FUNCTION_BLOCK TcoContext_App_1 EXTENDS TcoContext
VAR_INPUT
END_VAR
VAR_OUTPUT
END_VAR
VAR
	ResetToZero : BOOL := TRUE;
	C1	:	LINT	:= 100;
	C2	:	LINT	:= 200;
	TcoObject_Counter_1 : TcoObject_Counter(THIS^);
	TcoObject_Counter_2 : TcoObject_Counter(THIS^);
	Cycle	:	LINT:=-1;
	TcoTask_DownCounter_1	: TcoTask_DownCounter(THIS^);
	TcoTask_DownCounter_2	: TcoTask_DownCounter(THIS^);
	TcoObject_Counter_1_CountUp_Done_RTRIG : R_TRIG;
	TcoObject_Counter_1_CountDown_Done_RTRIG : R_TRIG;
	TcoObject_Counter_2_CountUp_Done_RTRIG : R_TRIG;
	TcoObject_Counter_2_CountDown_Done_RTRIG : R_TRIG;
	TcoObject_Counter_1_CountUp_Reset : BOOL;
	TcoObject_Counter_1_CountDown_Reset : BOOL;
	TcoObject_Counter_2_CountUp_Reset : BOOL;
	TcoObject_Counter_2_CountDown_Reset : BOOL;
END_VAR

METHOD PROTECTED  Main
//VAR
//	state : TcoState(THIS^,false); 
//END_VAR
//TcoTaskInvokeLevel();
//TcoTaskInvokeImpulse();
TcoTaskInvokeReset();
//state.Restore(TcoObject_Counter_1.TcoTask_CountUp).Restore(TcoObject_Counter_2.TcoTask_CountUp);

TcoTaskImplementation();
END_METHOD

METHOD TcoTaskImplementation
VAR_INPUT
END_VAR
THIS^.TcoTask_DownCounter_1();
//Init Invoke
IF THIS^.TcoTask_DownCounter_1.CounterValue = -1 THEN
	THIS^.TcoTask_DownCounter_1.SetUpValue := C1;
	THIS^.TcoTask_DownCounter_1.Invoke();
END_IF
//Next Invoke during execution
IF	THIS^.TcoTask_DownCounter_1.InTheMiddle THEN
	THIS^.TcoTask_DownCounter_1.SetUpValue := 2 * THIS^.TcoTask_DownCounter_1.SetUpValue;
	THIS^.TcoTask_DownCounter_1.Invoke();
END_IF
//Done and Invoke again
IF THIS^.TcoTask_DownCounter_1.Done THEN
	THIS^.TcoTask_DownCounter_1.SetUpValue := C1;
	THIS^.TcoTask_DownCounter_1.Invoke();
END_IF

THIS^.TcoTask_DownCounter_2();
//Init Invoke
IF THIS^.TcoTask_DownCounter_2.CounterValue = -1 THEN
	THIS^.TcoTask_DownCounter_2.SetUpValue := C2;
	THIS^.TcoTask_DownCounter_2.Invoke();
END_IF
//Next Invoke during execution
IF	THIS^.TcoTask_DownCounter_2.InTheMiddle THEN
	THIS^.TcoTask_DownCounter_2.SetUpValue := 2 * THIS^.TcoTask_DownCounter_2.SetUpValue;
	THIS^.TcoTask_DownCounter_2.Invoke();
END_IF
//Done and Invoke again
IF THIS^.TcoTask_DownCounter_2.Done THEN
	THIS^.TcoTask_DownCounter_2.SetUpValue := C2;
	THIS^.TcoTask_DownCounter_2.Invoke();
END_IF
END_METHOD

METHOD TcoTaskInvokeImpulse
VAR_INPUT
END_VAR
TcoObject_Counter_1();

TcoObject_Counter_2();

TcoObject_Counter_1_CountUp_Done_RTRIG(CLK := THIS^.TcoObject_Counter_1.TcoTask_CountUp.Done );
TcoObject_Counter_1_CountDown_Done_RTRIG(CLK := THIS^.TcoObject_Counter_1.TcoTask_CountDown.Done );
TcoObject_Counter_2_CountUp_Done_RTRIG(CLK := THIS^.TcoObject_Counter_2.TcoTask_CountUp.Done );
TcoObject_Counter_2_CountDown_Done_RTRIG(CLK := THIS^.TcoObject_Counter_2.TcoTask_CountDown.Done );


IF ResetToZero THEN
	THIS^.TcoObject_Counter_1.TcoTask_ResetToZero.Invoke();
	THIS^.TcoObject_Counter_2.TcoTask_ResetToZero.Invoke();
	ResetToZero := FALSE;
END_IF

IF THIS^.TcoObject_Counter_1.TcoTask_ResetToZero.Done THEN
	THIS^.TcoObject_Counter_1.StartCountUp(C1);
	THIS^.TcoObject_Counter_1.TcoTask_ResetToZero.Restore();	//ResetToZeroTask has to be reseted, otherwise StartCountUp is called cyclically
END_IF;

IF THIS^.TcoObject_Counter_2.TcoTask_ResetToZero.Done THEN
	THIS^.TcoObject_Counter_2.StartCountUp(C2);
	THIS^.TcoObject_Counter_2.TcoTask_ResetToZero.Restore(); //ResetToZeroTask has to be reseted, otherwise StartCountUp is called cyclically
END_IF;

IF TcoObject_Counter_1_CountUp_Done_RTRIG.Q THEN
	THIS^.TcoObject_Counter_1.StartCountDown(-C1);
END_IF;

IF TcoObject_Counter_2_CountUp_Done_RTRIG.Q THEN
	THIS^.TcoObject_Counter_2.StartCountDown(-C2);
END_IF;

IF THIS^.TcoObject_Counter_1.TcoTask_CountDown.Done AND NOT THIS^.TcoObject_Counter_1.TcoTask_CountUp.Busy
	AND THIS^.TcoObject_Counter_2.TcoTask_CountDown.Done AND NOT THIS^.TcoObject_Counter_2.TcoTask_CountUp.Busy THEN
	THIS^.TcoObject_Counter_1.StartCountUp(C1);
	THIS^.TcoObject_Counter_2.StartCountUp(C2);
END_IF

Cycle	:= THIS^.TcoObject_Counter_2.Cycle ;
END_METHOD

METHOD TcoTaskInvokeLevel
VAR_INPUT
END_VAR
TcoObject_Counter_1();

TcoObject_Counter_2();

IF ResetToZero THEN
	THIS^.TcoObject_Counter_1.TcoTask_ResetToZero.Invoke();
	THIS^.TcoObject_Counter_2.TcoTask_ResetToZero.Invoke();
	ResetToZero := FALSE;
END_IF

IF THIS^.TcoObject_Counter_1.TcoTask_ResetToZero.Done THEN
	THIS^.TcoObject_Counter_1.StartCountUp(C1);
	THIS^.TcoObject_Counter_1.TcoTask_ResetToZero.Restore();	//ResetToZeroTask has to be reseted, otherwise StartCountUp is called cyclically
END_IF;

IF THIS^.TcoObject_Counter_1.TcoTask_CountUp.Done THEN
	THIS^.TcoObject_Counter_1.StartCountDown(-C1);
END_IF;

IF THIS^.TcoObject_Counter_2.TcoTask_ResetToZero.Done THEN
	THIS^.TcoObject_Counter_2.StartCountUp(C2);
	THIS^.TcoObject_Counter_2.TcoTask_ResetToZero.Restore(); //ResetToZeroTask has to be reseted, otherwise StartCountUp is called cyclically
END_IF;

IF THIS^.TcoObject_Counter_2.TcoTask_CountUp.Done THEN
	THIS^.TcoObject_Counter_2.StartCountDown(-C2);
END_IF;

IF THIS^.TcoObject_Counter_1.TcoTask_CountDown.Done AND THIS^.TcoObject_Counter_2.TcoTask_CountDown.Done THEN
	THIS^.TcoObject_Counter_1.StartCountUp(C1);
	THIS^.TcoObject_Counter_2.StartCountUp(C2);
END_IF

Cycle	:= THIS^.TcoObject_Counter_2.Cycle ;
END_METHOD

METHOD TcoTaskInvokeReset
VAR_INPUT
END_VAR
TcoObject_Counter_1();

TcoObject_Counter_2();

TcoObject_Counter_1_CountUp_Reset 	:= FALSE;
TcoObject_Counter_1_CountDown_Reset := False;
TcoObject_Counter_2_CountUp_Reset 	:= False;
TcoObject_Counter_2_CountDown_Reset := False;

THIS^.TcoObject_Counter_1.TcoTask_ResetToZero.Invoke();
THIS^.TcoObject_Counter_2.TcoTask_ResetToZero.Invoke();
THIS^.TcoObject_Counter_1.StartCountUp(C1);
THIS^.TcoObject_Counter_1.StartCountDown(-C1);
THIS^.TcoObject_Counter_2.StartCountUp(C2);
THIS^.TcoObject_Counter_2.StartCountDown(-C2);

IF THIS^.TcoObject_Counter_1.TcoTask_CountUp.Busy THEN
	THIS^.TcoObject_Counter_1.TcoTask_CountDown.Restore();
	TcoObject_Counter_1_CountDown_Reset := TRUE;
END_IF

IF THIS^.TcoObject_Counter_2.TcoTask_CountUp.Busy THEN
	THIS^.TcoObject_Counter_2.TcoTask_CountDown.Restore();
	TcoObject_Counter_2_CountDown_Reset := TRUE;
END_IF

IF THIS^.TcoObject_Counter_2.TcoTask_CountDown.Busy THEN
	THIS^.TcoObject_Counter_1.TcoTask_CountUp.Restore();
	TcoObject_Counter_1_CountUp_Reset := TRUE;
END_IF


IF THIS^.TcoObject_Counter_2.TcoTask_CountDown.Busy THEN
	THIS^.TcoObject_Counter_2.TcoTask_CountUp.Restore();
	TcoObject_Counter_2_CountUp_Reset := TRUE;
END_IF

Cycle	:= THIS^.TcoObject_Counter_2.Cycle ;
END_METHOD

END_FUNCTION_BLOCK

(* stored: Version 1.1.0.1, ProductVersion 3.1.4024.6
   POU TcoContext_App_1: Id {4453eacb-a9a5-41b5-b0f4-727cecf60f7b}, SpecialFunc None
   Method Main: Id {5016e8d2-ba57-4ab2-8cd2-2579f738e57b}
   Method TcoTaskImplementation: Id {dafc2e8f-8fa8-481c-af67-05d32184381c}
   Method TcoTaskInvokeImpulse: Id {2d7a306c-08a8-4b1c-b614-8726f75ef05c}
   Method TcoTaskInvokeLevel: Id {dc70d169-5114-4e96-8922-96973420284b}
   Method TcoTaskInvokeReset: Id {22abd949-3f5f-4a27-8dcb-dad4f646b374} *)
